FUNCTION_BLOCK TechnologicalDataManager EXTENDS TcoData.TcoDataExchange
VAR
    _data : TechnologyData := (Parent := THIS^);
END_VAR

SUPER^();

PROPERTY Data : REFERENCE TO TechnologyData
GET
Data REF= _data;
END_GET
END_PROPERTY

END_FUNCTION_BLOCK

(* stored: Version 1.1.0.1
   POU TechnologicalDataManager: Id {06b46b93-bcf9-022c-0edf-e96bd18e6660}, SpecialFunc None
   Property Data: Id {61dc4c74-76bd-0bcc-1193-82087be92c90}
   Get Get: Id {9c2f366a-846c-0abb-3224-43f8841e354b} *)
